// TIA Portal project "ejemplo0506_introaTIA" (V20)

(* hardware
DEVICE "S7-1200 station_1"  S7-1200 Station
   slot 0: "Rack_0"  S7-1200 Rack  Rack  V1.0
   slot 1: "PLC_1"  CPU 1215C AC/DC/Rly  6ES7 215-1BG40-0XB0  V4.7
*)

// ===== PLC "PLC_1"  CPU 1215C AC/DC/Rly =====

VAR_GLOBAL   // PLC tag table "Default tag table"
   "Start I" AT %I0.0 : Bool;
   "K1" AT %Q0.0 : Bool;
   "Etapa 1" AT %M0.0 : Bool;
   "Etapa 2" AT %M0.1 : Bool;
   "Etapa 3" AT %M0.2 : Bool;
   "Etapa 4" AT %M0.3 : Bool;
   "K2" AT %Q0.1 : Bool;
   "Tag_1" AT %M10.0 : Bool;
END_VAR

// folder: System blocks/Program resources

DATA_BLOCK "IEC_Timer_0_DB"   // DB1
{ S7_Optimized_Access := 'TRUE' }
AUTHOR : Simatic
FAMILY : IEC
NAME : IEC_TMR
VERSION : 1.0
// stored: InstanceOfName IEC_TIMER
"IEC_TIMER"
BEGIN
END_DATA_BLOCK

// folder: (top level)

ORGANIZATION_BLOCK "Main"   // OB1, LAD, ProgramCycle
TITLE = "Main Program Sweep (Cycle)"
{ S7_Optimized_Access := 'TRUE' }
VERSION : 0.1
   VAR_INPUT
      Initial_Call : Bool;   // Initial call of this OB
      Remanence : Bool;   // =True, if remanent data are available
   END_VAR
BEGIN

REGION Network 1: Etapa 1
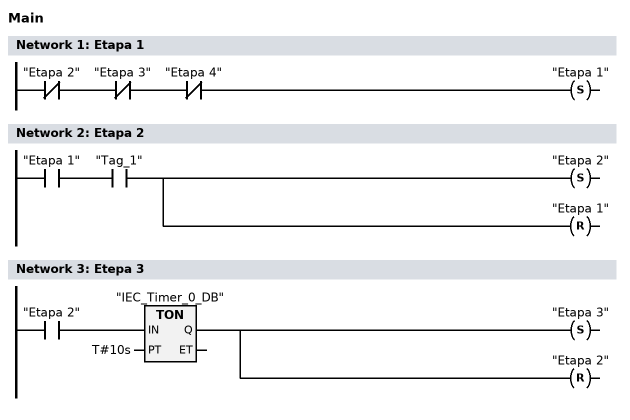
   RUNG wire#powerrail
      I_Contact( "Etapa 2" )
      I_Contact( "Etapa 3" )
      I_Contact( "Etapa 4" )
      S_Coil( "Etapa 1" )
   END_RUNG
   // the same network as SCL:
   IF NOT "Etapa 2" AND NOT "Etapa 3" AND NOT "Etapa 4" THEN "Etapa 1" := TRUE; END_IF;
END_REGION

REGION Network 2: Etapa 2
   RUNG wire#powerrail
      Contact( "Etapa 1" )
      Contact( "Tag_1" )
      wire#w1
      S_Coil( "Etapa 2" )
   END_RUNG
   RUNG wire#w1
      R_Coil( "Etapa 1" )
   END_RUNG
   // the same network as SCL:
   IF "Etapa 1" AND "Tag_1" THEN
       "Etapa 2" := TRUE;
       "Etapa 1" := FALSE;
   END_IF;
END_REGION

REGION Network 3: Etepa 3
   "IEC_Timer_0_DB".TON(IN := "Etapa 2", PT := T#10s);
   IF "IEC_Timer_0_DB".Q THEN
       "Etapa 3" := TRUE;
       "Etapa 2" := FALSE;
   END_IF;
END_REGION
END_ORGANIZATION_BLOCK